(* PLC project Generated.project, CODESYS CODESYS V3.5 SP19 Patch 1 *)
(* stored: creationDateTime 2026-08-11T14:02:33.668053, modificationDateTime 2026-08-11T14:02:33.668053 *)

(* ═══════════════════════════════════════════════════════════════ 🔧 ST_BypassTranslation — Bypass maintenance dédiés à Translation M3 ─────────────────────────────────────────────────────────────── 🔒 Doctrine : actionnable UNIQUEMENT en MAINT_N2, RETAIN, jamais masque les autres défauts du même bloc (voir REGISTRE_ACTIONS_Bypass_v1.0 (archive)). ═══════════════════════════════════════════════════════════════ *)
TYPE ST_BypassTranslation : STRUCT
  OperatorComm : BOOL;  (* 📡 1. Communication & Systèmes auxiliaires 📡 Bypass communication esclave CANopen Joystick / heartbeat IHM *)
  DriveComm : BOOL;  (* 📡 Bypass diagnostic esclave EtherCAT AC600 (variateur) *)
  ContactorFeedback : BOOL;  (* 🔌 Bypass feedbacks contacteur de frein *)
  PhaseRotation : BOOL;  (* ⚡ Bypass défaut rotation de phases (commun machine) *)
  BrakeThermal : BOOL;  (* 🌡️ Bypass surchauffe thermique frein (commun machine) *)
  LimitSwitch : BOOL;  (* 🚧 2. Limites physiques et Positionnement 🚧 Bypass fins de course physiques avant/arrière *)
  SensorIncoherent : BOOL;  (* 🧭 Bypass incohérence mot capteurs de position *)
  MinHeight : BOOL;  (* 🆕 2026-08-06 : Bypass interlock hauteur mini M1/M2 requise pour translation *)
  MecaA : BOOL;  (* ⚙️ 3. Sécurité Mécanique (Méca A-B) 🔄 Bypass Méca A : mouvement non commandé à l'arrêt *)
  MecaB : BOOL;  (* 🛑 Bypass Méca B : absence confirmation arrêt (frein/contacteurs) *)
  Safety : BOOL;  (* 🛡️ 4. Hiérarchie & Restauration 🛡️ Bypass groupé : tous les bits qui provoquent un PowerCutOff *)
  Process : BOOL;  (* ⚙️ Bypass groupé : tous les bits qui provoquent un SafeStop *)
  Global : BOOL;  (* 🌐 Bypass Global : ignore toutes les sécurités de cet axe *)
  Initialized : BOOL := FALSE;  (* 🐛 FIX persistance (voir DOC/AUDITS/ConfigPersistence/) : flag restauration boot dédié (défaut FALSE non ambigu, contrairement à une valeur métier) — PRG_SUPERVISION_CFC.st 🚦 TRUE = bypass restauré depuis GVL_BypassRetain ce boot *)
END_STRUCT;
END_TYPE
